TYPE csp_case_feed_phase_status_enum :
(		
	CSP_CASE_FEED_STATUS_PHASE_START						:= 0,
	CSP_CASE_FEED_STATUS_PHASE_DISABLE 						:= 10,
	CSP_CASE_FEED_STATUS_PHASE_ENABLE 						:= 20,	
	CSP_CASE_FEED_STATUS_PHASE_ACTIVATE_KINEMATIC			:= 30,
	CSP_CASE_FEED_STATUS_PHASE_CALCULATE_SLAVE_POSITION		:= 40,
	CSP_CASE_FEED_STATUS_PHASE_READ_SLAVE_POSITION			:= 50,	
	CSP_CASE_FEED_STATUS_PHASE_CHECK_Y_POS					:= 51,
	CSP_CASE_FEED_STATUS_PHASE_WAIT_FOR_FOLL_SPREAD			:= 52,
	CSP_CASE_FEED_STATUS_PHASE_MOVE_SLAVE_POSITION			:= 60,
	CSP_CASE_FEED_STATUS_PHASE_MOVED_SLAVE_POSITION			:= 70,
	CSP_CASE_FEED_STATUS_PHASE_DONE 						:= 900,
	CSP_CASE_FEED_STATUS_PHASE_ERROR 						:= 999
) := CSP_CASE_FEED_STATUS_PHASE_START;
END_TYPE

(* stored: Version 1.1.0.1, ProductVersion 3.1.4024.3
   DUT csp_case_feed_phase_status_enum: Id {b8021630-cbc4-444b-8cda-9df0043acec4} *)
